Fanuc KAREL source: KA00101.KL

PROGRAM KA00101
%NOLOCKGROUP
VAR
  SRC: VECTOR
  DST: POSITION
BEGIN
  SRC.X = 1.0
  DST = SRC
END KA00101
